TYPE Vision_IO_typ:
STRUCT
	Inputs	: Vision_Inputs_typ;
	Outputs	: Vision_Outputs_typ;
END_STRUCT
END_TYPE

(* stored: Version 1.1.0.1, ProductVersion 3.1.4024.12
   DUT Vision_IO_typ: Id {96fa3846-8f93-0bdc-263b-8cf55dbbbf55} *)
